// Mitsubishi GX Works2 project: 4   PLC: FX3U/FX3UC

PROGRAM MAIN
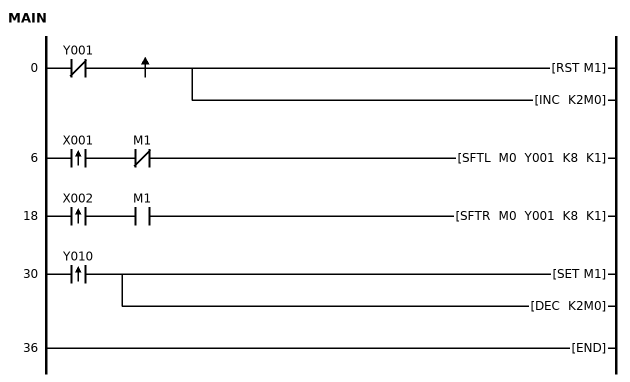
0     LDI     Y001
      MEP
      RST     M1
      INC     K2M0
6     LDP     X001
      ANI     M1
      SFTL    M0 Y001 K8 K1
18    LDP     X002
      AND     M1
      SFTR    M0 Y001 K8 K1
30    LDP     Y010
      SET     M1
      DEC     K2M0
36    END
END_PROGRAM
